Omron CX-Programmer project NewProject (CX-Programmer 9.75)

# PLC OMRON: CP1E N30

## Global symbols (name address type ; comment)
T000 BOOL  ; T0
T001 BOOL  ; T1

## Program NewProgram1 (cyclic task 0)
Local symbols
Lamp 100.00 BOOL  ; 100.00
PB 0.00 BOOL  ; 0.00
PB1 0.01 BOOL  ; 0.01

### Section Section1

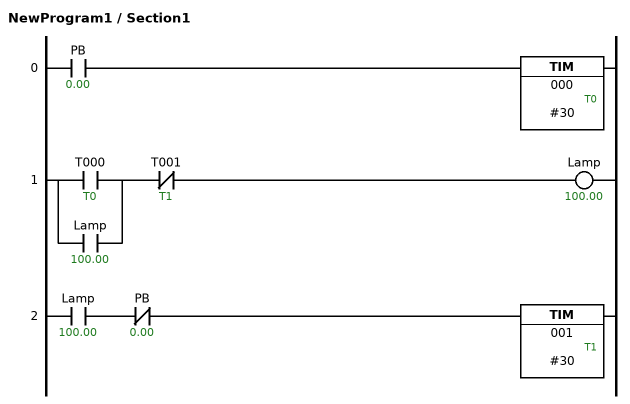
; rung 0
LD PB  ; 0.00
TIM 000 #30  ; T0
; rung 1
LD T000  ; T0
OR Lamp  ; 100.00
ANDNOT T001  ; T1
OUT Lamp  ; 100.00
; rung 2
LD Lamp  ; 100.00
ANDNOT PB  ; 0.00
TIM 001 #30  ; T1

### Section END
; rung 0
END(001)